(*
Nazwa:			FB_RgbLedTape
Opis:			Sterowanie taśmamy przez moduł sterownika EL6851
Wersja:			v0.2
Data:			2024-03-13
Autor:			AM,DP
Urzadzenia:		EL6851
Konfiguracja:	GVL_DMX z aProcessData
Info:
Zmiany:
- 20240318 [DP] Dodanie migajacych dwóch kolorów na przemian
*)
FUNCTION_BLOCK FB_RgbLedTape_EL2563

VAR_INPUT
	
	bEnable					:		BOOL;	
	nCh1Red					:		INT;
	nCh2Green				:		INT;
	nCh3Blue				:		INT;
	nCh4White				:		INT;
	nCh5Reserve				:		INT;
	
	bBlink					:		BOOL;
	bBlink2Colors			:		BOOL;	
	nDelayBlink				:		INT :=5;
	nMaxBlinkValue			:		INT:=16000;	

	nMinBlinkValue			:		INT:=2000;	
END_VAR

VAR_OUTPUT
END_VAR

VAR_IN_OUT
	AiProcessData			   : ARRAY [1..5] OF INT;
END_VAR

VAR
	nCycleBlink			:	INT;	//Liczylnik cyklów dla tryby Migamie 
	nBlinkValue			:	INT;	//Biegle znaczenie dla migania
	bBlinkDir			:	BOOL; 	//kierunek (zmieńszenie/zwiękzenie nBlinkValue)
	bChangeColor: BOOL;
	iBlink2ColorsCase: INT;
	toniBlink2ColorsCase: TON;
END_VAR

IF (bEnable) THEN
	IF (bBlink2Colors) THEN
		actBlink2Colors();
	ELSIF (bBlink) THEN
		actBlink();
	ELSE
		actNoBlink();
	END_IF
	
	
END_IF

ACTION actBlink:
IF (nCh1Red>0) THEN
	AiProcessData[1] := nBlinkValue;
ELSE
	AiProcessData[1] := 0;
END_IF

IF (nCh2Green>0) THEN
	AiProcessData[2] := nBlinkValue;
ELSE
	AiProcessData[2] := 0;
END_IF
	
IF (nCh3Blue>0) THEN
	AiProcessData[3] := nBlinkValue;
ELSE
	AiProcessData[3] := 0;
END_IF

IF (nCh4White>0) THEN
	AiProcessData[4] := nBlinkValue;
ELSE
	AiProcessData[4] := 0;
END_IF

IF (nCh5Reserve>0) THEN
	AiProcessData[5] := nBlinkValue;
ELSE
	AiProcessData[5] := 0;
END_IF

//Inc/dec dla nBlinkValue
nCycleBlink := nCycleBlink + 1;
IF (nCycleBlink > nDelayBlink) THEN
	
	//dodac
	IF (nBlinkValue < nMaxBlinkValue AND NOT bBlinkDir) THEN
		nBlinkValue :=nBlinkValue + 50;
		IF nBlinkValue < 0 THEN
		nBlinkValue := nMaxBlinkValue;
		bBlinkDir := TRUE;
		END_IF
	ELSE
		bBlinkDir := TRUE;
	END_IF
	
	//zwiększyć
	IF (nBlinkValue > nMinBlinkValue AND bBlinkDir) THEN
		nBlinkValue :=nBlinkValue - 100;
		IF nBlinkValue < 0 THEN
		nBlinkValue := nMinBlinkValue;
		bBlinkDir := FALSE;
		END_IF
	ELSE
		bBlinkDir := FALSE;
	END_IF
	
	nCycleBlink :=0;
END_IF
END_ACTION

ACTION actBlink2Colors:
bChangeColor;
toniBlink2ColorsCase(IN:=iBlink2ColorsCase=50,PT:=T#100MS);
CASE iBlink2ColorsCase OF
	0:
		AiProcessData[1] 	:= 0;
		AiProcessData[2] 	:= nCh2Green;
		AiProcessData[3] 	:= 0;
		AiProcessData[4] 	:= 0;
		
		iBlink2ColorsCase	:=	iBlink2ColorsCase	+	10;
		
	10:
		AiProcessData[2] := 	AiProcessData[2] - 50;
		IF 	AiProcessData[2] < 100 THEN
			iBlink2ColorsCase	:=	iBlink2ColorsCase	+	10;
		END_IF
		
	20:
		AiProcessData[3] 	:= 	AiProcessData[3] + 100;
		IF 	AiProcessData[3] > 32000 THEN
			iBlink2ColorsCase	:=	iBlink2ColorsCase	+	10;
		END_IF	

	30:
		AiProcessData[3] 	:= 	AiProcessData[3] - 100;
		IF 	AiProcessData[3] < 200 THEN
			iBlink2ColorsCase	:=	iBlink2ColorsCase	+	10;
		END_IF	
	
	40:
		AiProcessData[2] := 	AiProcessData[2] + 50;
		IF 	AiProcessData[2] > nCh2Green THEN
			iBlink2ColorsCase	:=	iBlink2ColorsCase	+	10;
		END_IF		
		
	50:
		IF toniBlink2ColorsCase.Q THEN
			iBlink2ColorsCase	:=	0;
		END_IF
END_CASE
END_ACTION

ACTION actNoBlink:
AiProcessData[1] :=nCh1Red;
AiProcessData[2] :=nCh2Green;
AiProcessData[3] :=nCh3Blue;
AiProcessData[4] :=nCh4White;
AiProcessData[5] :=nCh5Reserve;
END_ACTION

END_FUNCTION_BLOCK

(* stored: Version 1.1.0.1, ProductVersion 3.1.4026.13, FileIdentifier 89585761c9809b30b2cc69a54b90c529984a3321, FileSignature 0a0683ce6d5fbc8989b205e8c35dd4920dbb3aef240b28152f4f6a50915a730b8f5283582c741c4a3ae2ce011edfc92922dfe96764861baa8c198e3a120e2c2ea773849777fb41842e92526c81eb5f0748da4b7019d241d35a1adb1da87adb9aaa6ceaa5716a2a0be14008ff2ae85cb397655ef8fd4a55c74750b735725d78b9098141301494453e357c36f4c266dee2981481f538842c29541c7625726d2bc7db57560f7424697362ae5183c8f17bef82d00e1052b8a400a9dd09d4370cbbc0ddf39bf69c638add3a07efcd09297b9fc76e408fbca996443dc2423a6e033062e0b65fa52064f580679e4518ea4ef84472d8afa99d6b9ce62e2ca736f013a435
   POU FB_RgbLedTape_EL2563: Id {97535453-c227-42f1-8366-3de768a32b5d}, SpecialFunc None
   Action actBlink: Id {f868775f-d38d-4431-9524-6db15805ab60}
   Action actBlink2Colors: Id {b3f55fa6-7aa4-4619-a871-d225a3e6bc29}
   Action actNoBlink: Id {a18b904a-8569-4665-b6ca-ae530f67d9aa} *)
